FUNCTION_BLOCK FB_RoundBeltService EXTENDS FB_ActionBasic
VAR_INPUT
    xExecute      : BOOL;
    xAbort        : BOOL;
    TargetStation : INT;

    Cylinder : REFERENCE TO UNI_CylinderList;
    TimeOut  : LREAL := 90; // Unit : s
END_VAR
VAR_OUTPUT
    xAborted : BOOL;
    iErrorID : INT;
    ErrorMsg : STRING;
END_VAR
VAR
    StateBehavior   : CBML.ETrigATo;
    CurrentPosition : ST_PositionTable;
    CurrentData     : ARRAY[1..21] OF ST_PositionTable;
    uiCyclicStep    : UINT := 0;
    uiIndexLoop     : UINT;
	fbExecuteEdgeDetect :FB_EdgeDetect;
END_VAR

THIS^.IBehaviourModel := StateBehavior;
StateBehavior(xExecute := xExecute,
              xAbort := xAbort OR fbExecuteEdgeDetect.xFallingEdge,
              udiTimeOut := LREAL_TO_UDINT( TimeOut*1000000),
              xDone => xDone,
              xBusy => xBusy,
              xError => xError,
              xAborted => xAborted);

//Make sure that C# turns off execute to shut down the service
fbExecuteEdgeDetect(xInput :=xExecute);

//Error Msg
iErrorID := StateBehavior._model.iErrorID;
ErrorMsg := M_GetErrorMsg(xErrorID := iErrorID);

			  
A00_ReadPositionData();

ACTION A00_ReadPositionData:
FOR uiIndexLoop := 1 TO 20 DO
    CurrentData[uiIndexLoop] := FUN_GetPositionTableData(PositionName := 'B', Index := UINT_TO_LREAL(uiIndexLoop), Clip := E_ClipNo.A);
END_FOR
END_ACTION

METHOD CleanupAction
VAR_INPUT
    xAbortProposed : BOOL;
    iErrorIDProposed: INT;
END_VAR
VAR_OUTPUT
    xComplete : BOOL := TRUE;
    xAbort: BOOL := xAbortProposed;
 	iErrorID : INT := iErrorIDProposed;
END_VAR
uiCyclicStep := 0;
END_METHOD

METHOD CyclicAction
VAR_INPUT
    itfTimingController : CBML.ITimingController;
END_VAR
VAR_OUTPUT
    xComplete : BOOL := TRUE;
    iErrorID : INT := 0;
END_VAR
VAR_INST
	
END_VAR
xComplete := FALSE;
CASE uiCyclicStep OF
    0:
		//Check if current station is same as target
		IF ABS(CurrentPosition.X_Pos -  arAxisCtrl_gb[AxisNo.RoundBelt].Admin.Axis.NcToPlc.ModuloSetPos) < 0.2 THEN
			uiCyclicStep := 200;
			ELSE
			uiCyclicStep := 50;	
		END_IF
	50:
		// Retract all cylinders
        Cylinder.List.fbRoundBelt_ChargeZone_Plug.M_Retract();
        Cylinder.List.fbRoundBelt_TransmitCVZone_Plug.M_Retract();
        Cylinder.List.fbRoundBelt_WorkZone_Plug.M_Retract();
        Cylinder.List.fbRoundBelt_WorkZone_Press.M_Retract();

        IF Cylinder.List.fbRoundBelt_ChargeZone_Plug.InRearPosition AND
            Cylinder.List.fbRoundBelt_TransmitCVZone_Plug.InRearPosition AND
            Cylinder.List.fbRoundBelt_WorkZone_Plug.InRearPosition AND
            Cylinder.List.fbRoundBelt_WorkZone_Press.InRearPosition THEN
            uiCyclicStep := 100;
        END_IF
    100: 
	    // Move round belt to target station
        arAxisCtrl_gb[AxisNo.RoundBelt].PosMode.Position := CurrentPosition.X_Pos;
		 IF  arAxisCtrl_gb[AxisNo.RoundBelt].Admin.Axis.Status.Moving THEN
				uiCyclicStep := 190;
		 END_IF
		
	190:
        IF arAxisStatus_gb[AxisNo.RoundBelt].Admin._OpModeAck = ModePosAbs AND arAxisStatus_gb[AxisNo.RoundBelt].Admin.CmdDone AND
			(arAxisCtrl_gb[AxisNo.RoundBelt].Admin.Axis.Status.InTargetPosition OR arAxisCtrl_gb[AxisNo.RoundBelt].Admin.Axis.Status.Operational)
		THEN
            uiCyclicStep := 200;
        END_IF
	200:
        Cylinder.List.fbRoundBelt_ChargeZone_Plug.M_Extend();
        Cylinder.List.fbRoundBelt_TransmitCVZone_Plug.M_Extend();
        Cylinder.List.fbRoundBelt_WorkZone_Plug.M_Extend();
        

        IF Cylinder.List.fbRoundBelt_ChargeZone_Plug.InFrontPosition AND
            Cylinder.List.fbRoundBelt_TransmitCVZone_Plug.InFrontPosition AND
            Cylinder.List.fbRoundBelt_WorkZone_Plug.InFrontPosition THEN
            uiCyclicStep := 300;
        END_IF
	300:
		Cylinder.List.fbRoundBelt_WorkZone_Press.M_Extend();
		IF  Cylinder.List.fbRoundBelt_WorkZone_Press.InFrontPosition THEN
            xComplete := TRUE;
        END_IF
		//	xComplete := TRUE;
END_CASE

IF arAxisCtrl_gb[AxisNo.RoundBelt].Admin.Axis.Status.Error THEN
    iErrorID := 6; // Axis RoundBelt has error
END_IF

IF Cylinder.List.fbRoundBelt_ChargeZone_Plug.xError THEN
    iErrorID := 7;
END_IF

IF Cylinder.List.fbRoundBelt_TransmitCVZone_Plug.xError THEN
    iErrorID := 8;
END_IF

IF Cylinder.List.fbRoundBelt_WorkZone_Plug.xError THEN
    iErrorID := 9;
END_IF

IF Cylinder.List.fbRoundBelt_WorkZone_Press.xError THEN
    iErrorID := 10;
END_IF
END_METHOD

METHOD ExitAction
VAR_INPUT
    xAfterCleanup : BOOL;
    xInCopyCode : BOOL;
END_VAR
END_METHOD

METHOD M_GetErrorMsg : T_MaxString
VAR_INPUT
	xErrorID: INT;
END_VAR

VAR
	
END_VAR
CASE xErrorID OF
	0:
		M_GetErrorMsg := 'No Error';
	1:
		M_GetErrorMsg := 'Action time out';
	2:
		M_GetErrorMsg := 'Position Data invalid';
	3:
		M_GetErrorMsg := 'Index invalid';
	4:
		M_GetErrorMsg := 'Axis roundbelt not ready has Error';
	5:
		M_GetErrorMsg := 'Cylinder not ready has Error';
	6:
		M_GetErrorMsg := 'Axis RoundBelt has Error';
	7:
		M_GetErrorMsg := 'ChargeZone_Plug has Error';
	8:
		M_GetErrorMsg := 'TransmitCVZone_Plug has Error';
	9:
		M_GetErrorMsg := 'WorkZone_Plug has Error';
	10:
		M_GetErrorMsg := 'WorkZone_Press has Error';
END_CASE
END_METHOD

METHOD PRIVATE M_StationModify : BOOL
VAR_INPUT
	TargetStation : INT;
END_VAR

VAR_OUTPUT
	ModifiedTargetStation : INT;
END_VAR
ModifiedTargetStation := (TargetStation/2)+1;
END_METHOD

METHOD ResetAction
VAR_OUTPUT
    xComplete : BOOL := TRUE;
END_VAR
END_METHOD

METHOD StartAction
VAR_OUTPUT
    xComplete : BOOL := TRUE;
	iErrorID : INT := 0;
END_VAR

VAR
	ModifiedTargetPos : INT;
END_VAR
xComplete := FALSE;
M_StationModify(TargetStation,ModifiedTargetStation =>ModifiedTargetPos);
IF TargetStation >= 1 AND TargetStation <= 40 THEN
    CurrentPosition := CurrentData[ModifiedTargetPos];
ELSE
    iErrorID := 3; // Target Station invalid.
    RETURN;
END_IF
uiCyclicStep := 0;

IF arAxisCtrl_gb[AxisNo.RoundBelt].Admin.Axis.Status.NotMoving AND
    NOT arAxisCtrl_gb[AxisNo.RoundBelt].Admin.Axis.Status.Error THEN
    xComplete := TRUE;
ELSE
    iErrorID := 4; // Axis not ready
END_IF

//IF Cylinder.List.fbRoundBelt_ChargeZone_Plug.xBusy AND Cylinder.List.fbRoundBelt_TransmitCVZone_Plug.xBusy AND 
//	Cylinder.List.fbRoundBelt_WorkZone_Plug.xBusy AND Cylinder.List.fbRoundBelt_WorkZone_Press.xBusy AND NOT 
//	Cylinder.List.fbRoundBelt_ChargeZone_Plug.xError AND NOT Cylinder.List.fbRoundBelt_TransmitCVZone_Plug.xError
//	AND NOT Cylinder.List.fbRoundBelt_WorkZone_Plug.xError AND NOT Cylinder.List.fbRoundBelt_WorkZone_Press.xError THEN
//	iErrorID := 5; // Cylinder not ready
//END_IF
xComplete := TRUE;
END_METHOD

END_FUNCTION_BLOCK

(* stored: Version 1.1.0.1, ProductVersion 3.1.4024.13
   POU FB_RoundBeltService: Id {8d75a2c3-8079-477f-bebf-e767c6ddb006}, SpecialFunc None
   Folder Action: Id {fb0ea1b7-3a55-401e-86f0-87cb968c2200}
   Folder Method: Id {a0cfead5-6aa1-458a-ab09-c8acb926f7c8}
   Action A00_ReadPositionData: Id {46cf0817-36b9-476c-9d1f-17310f877691}
   Method CleanupAction: Id {f6764331-1beb-4321-b18a-78b6014e8ed7}
   Method CyclicAction: Id {38f757a4-591e-49e8-b669-104182a2b01f}
   Method ExitAction: Id {944903a6-001d-4068-a074-95b113e1f2ad}
   Method M_GetErrorMsg: Id {1c95d7a3-dea2-43b7-8a85-ed4b935be22b}
   Method M_StationModify: Id {683ae689-c123-494d-8de1-cd4513cc4278}
   Method ResetAction: Id {acc22fc0-fafd-4f44-88d5-9cf0a6abebc3}
   Method StartAction: Id {bc4c5ba3-0601-41d1-a02e-4666588ee580} *)
